TYPE ST_HighTemperatureHeatingNetworkControl :
STRUCT
	fTargetTemperature : REAL;
	bAlgorithmPermission : BOOL;
END_STRUCT
END_TYPE

(* stored: Version 1.1.0.1, ProductVersion 3.1.4024.10
   DUT ST_HighTemperatureHeatingNetworkControl: Id {62265abc-da42-46bc-b58c-32abc31e7390} *)
